// TIA Portal V19 export
DATA_BLOCK "MANUAL TIME BASE DB"   // DB41
{ S7_Optimized_Access := 'TRUE' }
// stored: MemoryReserve 100
   VAR RETAIN
      "MFG VESSEL STIRRER RUN" : Struct
         SV : Int := 555;
         PV : Int := 0;
         "RESET TIME" : Bool := FALSE;
      END_STRUCT;
      "PREMIXING  VESSEL STIRRER RUN" : Struct
         SV : Int := 555;
         PV : Int := 0;
         "RESET TIME" : Bool := FALSE;
      END_STRUCT;
      "SUGAR VESSEL STIRRER RUN" : Struct
         SV : Int := 555;
         PV : Int := 0;
         "RESET TIME" : Bool := FALSE;
      END_STRUCT;
   END_VAR
BEGIN
END_DATA_BLOCK
